// TIA Portal V20 export
DATA_BLOCK "BK11"   // DB237
// stored: MemoryReserve 100
   VAR
      "X10-1 SIDE TAPING X-AXIS LIMIT SENSOR(-)" : Bool;
      "X11-1 SIDE TAPING X-AXIS LIMIT SENSOR(+)" : Bool;
      "X12-1 JR FIX STAGE X-AXIS LIMIT SENSOR(-)" : Bool;
      "X13-1 JR FIX STAGE X-AXIS LIMIT SENSOR(+)" : Bool;
      "X14-1 JR FIX STAGE C-AXIS LIMIT SENSOR(-)" : Bool;
      "X15-1 JR FIX STAGE C-AXIS LIMIT SENSOR(+)" : Bool;
      "X16-1 STACK DETECT SENSOR" : Bool;
      "X17-1 SIDE TAPE FIX STAGE OPEN" : Bool;
      "X10-2 SIDE TAPING X-AXIS HOME SENSOR" : Bool;
      "X11-2 SPARE" : Bool;
      "X12-2 JR FIX STAGE X-AXIS HOMING SENSOR" : Bool;
      "X13-2 SPARE" : Bool;
      "X14-2 JR FIX STAGE X-AXIS HOMING SENSOR" : Bool;
      "X15-2 SPARE" : Bool;
      "X16-2 SIDE TAPE CLAMP SAFETY PIN LOADING SENSOR" : Bool;
      "X17-2 SIDE TAPE FIX STAGE CLOSE" : Bool;
   END_VAR
BEGIN
END_DATA_BLOCK
